TYPE ST_Robot_Mitsubishi_Packet_2012 :
STRUCT
	// Packet number - 2012.
	// To robot.
	// Robot cycle control packet.
	// Trigger.
	
	Header							: DINT := 2012;													// Packet header.
	
	TargetState						: DINT;															// 0 for cycle End, 1 for cycle Start.
	
END_STRUCT
END_TYPE

(* stored: Version 1.1.0.1, ProductVersion 3.1.4024.2
   DUT ST_Robot_Mitsubishi_Packet_2012: Id {ef3e5c45-1576-4887-a644-a04b57a2a96d} *)
